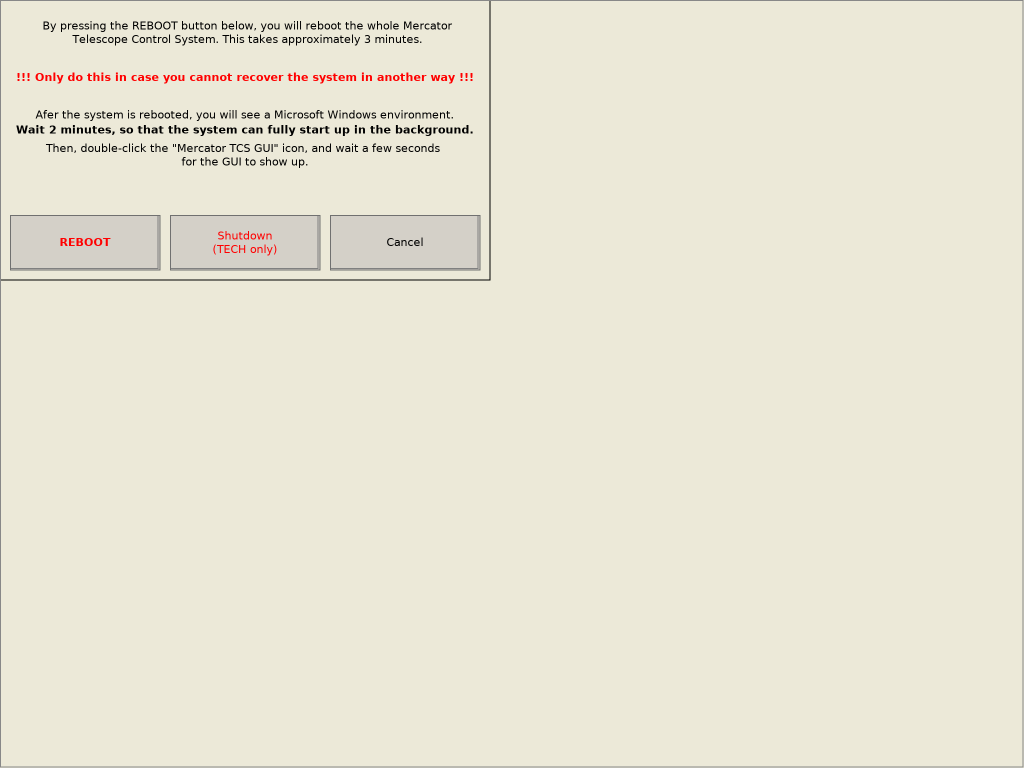
VISUALIZATION VISU_MTCSRebootDialog  // 1024x768
    Rectangle (0,0 490x280)
    Rectangle (0,5 495x55), "By pressing the REBOOT button below, you will reboot the whole Mercator Telescope Control System. This takes approximately 3 minutes."
    Rectangle (0,105 490x20), "Afer the system is rebooted, you will see a Microsoft Windows environment."
    Rectangle (0,120 490x20), "Wait 2 minutes, so that the system can fully start up in the background."
    Rectangle (0,135 490x40), "Then, double-click the "Mercator TCS GUI" icon, and wait a few seconds for the GUI to show up."
    Rectangle (0,50 490x55), "!!! Only do this in case you cannot recover the system in another way !!!"
    Button (10,215 150x55), "REBOOT", input disabled if: GLOBAL.mtcs.processes.reboot.statuses.enabledStatus.disabled
        OnMouseClick: execute { GLOBAL.mtcs.processes.reboot.do_request := TRUE; }
    Button (330,215 150x55), "Cancel"
        OnMouseClick: CloseDialog Dialog=VISU_MTCSRebootDialog, Result=Cancel, NumpadKeypadSet=True
    Button (170,215 150x55), "Shutdown (TECH only)", input disabled if: GLOBAL.mtcs.processes.shutdown.statuses.enabledStatus.disabled
        OnMouseClick: execute { GLOBAL.mtcs.processes.shutdown.do_request := TRUE; }
END_VISUALIZATION

(* stored: Version 1.1.0.1, ProductVersion 3.1.4018.5
   Visu VISU_MTCSRebootDialog: Id {3503e0a2-f61e-40d4-bb69-22b575bd1506} *)
